// TIA Portal V18 export
// export: Created 2025-12-01T17:51:05.437198Z, ExportSetting None, DisplayName Totally Integrated Automation Portal, DisplayVersion V18 Update 5, DisplayName TIA Portal Openness, DisplayVersion V18 Update 5, DisplayName TIA Portal Teamcenter Gateway, DisplayVersion V18, DisplayName TIA Portal Version Control Interface, DisplayVersion V18, DisplayName STEP 7 Professional, DisplayVersion V18 Update 5, DisplayName STEP 7 Safety, DisplayVersion V18, DisplayName WinCC Professional, DisplayVersion V18 Update 5
FUNCTION "ST10Cyl_interface51-60" : Void   // FC1025, LAD
{ S7_Optimized_Access := 'FALSE' }
// stored: AutoNumber false, SetENOAutomatically false
   VAR_INPUT
      AlwaysON : Bool;
      E_stop : Bool;
   END_VAR
   VAR_TEMP
      tTest : Bool;
   END_VAR
   VAR_TEMP   // added for the SCL form of the ladder/FBD networks
      _w1 : Bool;
   END_VAR
BEGIN

REGION Network 1 (SCL): Cylinder 51-60 IO Interface (SCL)

   //Cylinder51 IO  L-UnloadingTransCylinder
   //Input
   "ST10Cylinder".Cy[51].In.WorkPositionSensor := "iL-UnloadingTransCylinderInWP";
   "ST10Cylinder".Cy[51].In.HomePositionSensor := "iL-UnloadingTransCylinderInHP";
   //Output
   "oL-UnloadingTransCylinderToWP" := "ST10Cylinder".Cy[51].Out.GoWorkPosition;
   "oL-UnloadingTransCylinderToHP" := "ST10Cylinder".Cy[51].Out.GoHomePosition;

   //Cylinder52 IO  L-UnloadingTransPalletLocationCylinder
   //Input
   "ST10Cylinder".Cy[52].In.WorkPositionSensor := "iL-UnloadingTransPalletLocationCylinderInWP";
   "ST10Cylinder".Cy[52].In.HomePositionSensor := "iL-UnloadingTransPalletLocationCylinderInHP";
   //Output
   "oL-UnloadingTransPalletLocationCylinderToWP" := "ST10Cylinder".Cy[52].Out.GoWorkPosition;
   "oL-UnloadingTransPalletLocationCylinderToHP" := "ST10Cylinder".Cy[52].Out.GoHomePosition;

   //Cylinder53 IO  L-UnloadingStopperCylinder1
   //Input
   "ST10Cylinder".Cy[53].In.WorkPositionSensor := "oL-UnloadingStopperCylinder1_ToWP";
   "ST10Cylinder".Cy[53].In.HomePositionSensor := "oL-UnloadingStopperCylinder1_ToHP";
   //Output
   "oL-UnloadingStopperCylinder1_ToWP" := "ST10Cylinder".Cy[53].Out.GoWorkPosition;
   "oL-UnloadingStopperCylinder1_ToHP" := "ST10Cylinder".Cy[53].Out.GoHomePosition;

   //Cylinder54 IO  L-UnloadingStopperCylinder2
   //Input
   "ST10Cylinder".Cy[54].In.WorkPositionSensor := "oL-UnloadingStopperCylinder2_ToWP";
   "ST10Cylinder".Cy[54].In.HomePositionSensor := "oL-UnloadingStopperCylinder2_ToHP";
   //Output
   "oL-UnloadingStopperCylinder2_ToWP" := "ST10Cylinder".Cy[54].Out.GoWorkPosition;
   "oL-UnloadingStopperCylinder2_ToHP" := "ST10Cylinder".Cy[54].Out.GoHomePosition;

   //Cylinder55 IO  L-UnloadingStopperCylinder3
   //Input
   "ST10Cylinder".Cy[55].In.WorkPositionSensor := "oL-UnloadingStopperCylinder3_ToWP";
   "ST10Cylinder".Cy[55].In.HomePositionSensor := "oL-UnloadingStopperCylinder3_ToHP";
   //Output
   "oL-UnloadingStopperCylinder3_ToWP" := "ST10Cylinder".Cy[55].Out.GoWorkPosition;
   "oL-UnloadingStopperCylinder3_ToHP" := "ST10Cylinder".Cy[55].Out.GoHomePosition;

   (*
   //Cylinder56  L-UnloadingStopperCylinder2_2
   //Input
   "ST10Cylinder".Cy[56].In.WorkPositionSensor := "oL-UnloadingStopperCylinder2_2";
   "ST10Cylinder".Cy[56].In.HomePositionSensor := NOT "oL-UnloadingStopperCylinder2_2";
   //Output
   "oL-UnloadingStopperCylinder2_2" := "ST10Cylinder".Cy[56].Out.GoWorkPosition;
   //"oI-0080TrayLoadingTraySupportCylinder1ToHP" := "ST10Cylinder".Cy[56].Out.GoHomePosition;

   //Cylinder57 L-UnloadingStopperCylinder3_1
   //Input
   "ST10Cylinder".Cy[57].In.WorkPositionSensor := "oL-UnloadingStopperCylinder3_1";
   "ST10Cylinder".Cy[57].In.HomePositionSensor := NOT "oL-UnloadingStopperCylinder3_1";
   //Output
   "oL-UnloadingStopperCylinder3_1" := "ST10Cylinder".Cy[57].Out.GoWorkPosition;
   //"oI-0070TrayLoadingTraySupportCylinder8ToHP" := "ST10Cylinder".Cy[57].Out.GoHomePosition;

   //Cylinder58 L-UnloadingStopperCylinder3_2
   //Input
   "ST10Cylinder".Cy[58].In.WorkPositionSensor := "oL-UnloadingStopperCylinder3_2";
   "ST10Cylinder".Cy[58].In.HomePositionSensor := NOT "oL-UnloadingStopperCylinder3_2";
   //Output
   "oL-UnloadingStopperCylinder3_2" := "ST10Cylinder".Cy[58].Out.GoWorkPosition;
   //"oI-0080TrayLoadingTrayLocationCylinderToHP" := "ST10Cylinder".Cy[58].Out.GoHomePosition;
   //

   *)
END_REGION

REGION Network 2: CY51 interface L-UnloadingTransCylinder
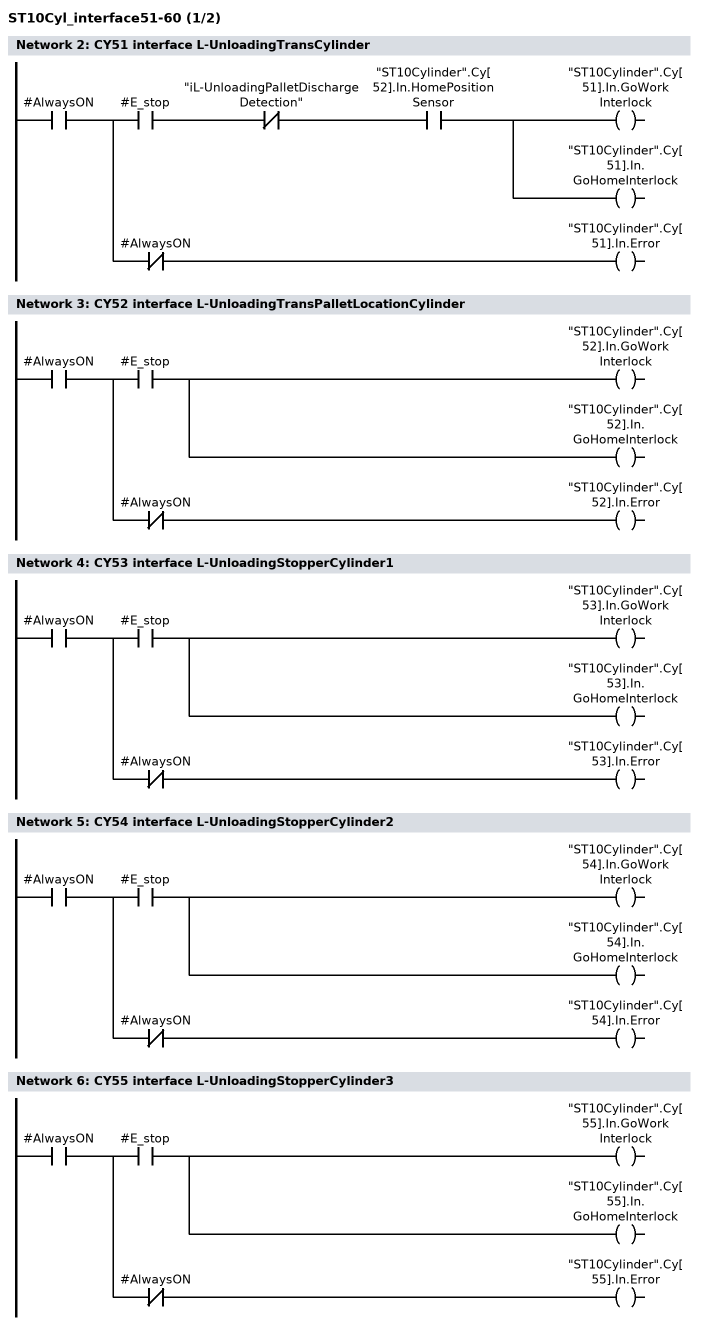
   RUNG wire#powerrail
      Contact( #AlwaysON )
      wire#w1
      Contact( #E_stop )
      I_Contact( "iL-UnloadingPalletDischargeDetection" )
      Contact( "ST10Cylinder".Cy[52].In.HomePositionSensor )
      wire#w2
      Coil( "ST10Cylinder".Cy[51].In.GoWorkInterlock )
   END_RUNG
   RUNG wire#w2
      Coil( "ST10Cylinder".Cy[51].In.GoHomeInterlock )
   END_RUNG
   RUNG wire#w1
      I_Contact( #AlwaysON )
      Coil( "ST10Cylinder".Cy[51].In.Error )
   END_RUNG
   // the same network as SCL:
   #_w1 := #AlwaysON AND #E_stop AND NOT "iL-UnloadingPalletDischargeDetection" AND "ST10Cylinder".Cy[52].In.HomePositionSensor;
   "ST10Cylinder".Cy[51].In.GoWorkInterlock := #AlwaysON AND #E_stop AND NOT "iL-UnloadingPalletDischargeDetection" AND "ST10Cylinder".Cy[52].In.HomePositionSensor;
   "ST10Cylinder".Cy[51].In.GoHomeInterlock := #_w1;
   "ST10Cylinder".Cy[51].In.Error := #AlwaysON AND NOT #AlwaysON;
END_REGION

REGION Network 3: CY52 interface L-UnloadingTransPalletLocationCylinder
   RUNG wire#powerrail
      Contact( #AlwaysON )
      wire#w1
      Contact( #E_stop )
      wire#w2
      Coil( "ST10Cylinder".Cy[52].In.GoWorkInterlock )
   END_RUNG
   RUNG wire#w2
      Coil( "ST10Cylinder".Cy[52].In.GoHomeInterlock )
   END_RUNG
   RUNG wire#w1
      I_Contact( #AlwaysON )
      Coil( "ST10Cylinder".Cy[52].In.Error )
   END_RUNG
   // the same network as SCL:
   "ST10Cylinder".Cy[52].In.GoWorkInterlock := #AlwaysON AND #E_stop;
   "ST10Cylinder".Cy[52].In.GoHomeInterlock := #AlwaysON AND #E_stop;
   "ST10Cylinder".Cy[52].In.Error := #AlwaysON AND NOT #AlwaysON;
END_REGION

REGION Network 4: CY53 interface L-UnloadingStopperCylinder1
   RUNG wire#powerrail
      Contact( #AlwaysON )
      wire#w1
      Contact( #E_stop )
      wire#w2
      Coil( "ST10Cylinder".Cy[53].In.GoWorkInterlock )
   END_RUNG
   RUNG wire#w2
      Coil( "ST10Cylinder".Cy[53].In.GoHomeInterlock )
   END_RUNG
   RUNG wire#w1
      I_Contact( #AlwaysON )
      Coil( "ST10Cylinder".Cy[53].In.Error )
   END_RUNG
   // the same network as SCL:
   "ST10Cylinder".Cy[53].In.GoWorkInterlock := #AlwaysON AND #E_stop;
   "ST10Cylinder".Cy[53].In.GoHomeInterlock := #AlwaysON AND #E_stop;
   "ST10Cylinder".Cy[53].In.Error := #AlwaysON AND NOT #AlwaysON;
END_REGION

REGION Network 5: CY54 interface L-UnloadingStopperCylinder2
   RUNG wire#powerrail
      Contact( #AlwaysON )
      wire#w1
      Contact( #E_stop )
      wire#w2
      Coil( "ST10Cylinder".Cy[54].In.GoWorkInterlock )
   END_RUNG
   RUNG wire#w2
      Coil( "ST10Cylinder".Cy[54].In.GoHomeInterlock )
   END_RUNG
   RUNG wire#w1
      I_Contact( #AlwaysON )
      Coil( "ST10Cylinder".Cy[54].In.Error )
   END_RUNG
   // the same network as SCL:
   "ST10Cylinder".Cy[54].In.GoWorkInterlock := #AlwaysON AND #E_stop;
   "ST10Cylinder".Cy[54].In.GoHomeInterlock := #AlwaysON AND #E_stop;
   "ST10Cylinder".Cy[54].In.Error := #AlwaysON AND NOT #AlwaysON;
END_REGION

REGION Network 6: CY55 interface L-UnloadingStopperCylinder3
   RUNG wire#powerrail
      Contact( #AlwaysON )
      wire#w1
      Contact( #E_stop )
      wire#w2
      Coil( "ST10Cylinder".Cy[55].In.GoWorkInterlock )
   END_RUNG
   RUNG wire#w2
      Coil( "ST10Cylinder".Cy[55].In.GoHomeInterlock )
   END_RUNG
   RUNG wire#w1
      I_Contact( #AlwaysON )
      Coil( "ST10Cylinder".Cy[55].In.Error )
   END_RUNG
   // the same network as SCL:
   "ST10Cylinder".Cy[55].In.GoWorkInterlock := #AlwaysON AND #E_stop;
   "ST10Cylinder".Cy[55].In.GoHomeInterlock := #AlwaysON AND #E_stop;
   "ST10Cylinder".Cy[55].In.Error := #AlwaysON AND NOT #AlwaysON;
END_REGION

REGION Network 7: CY56 interface
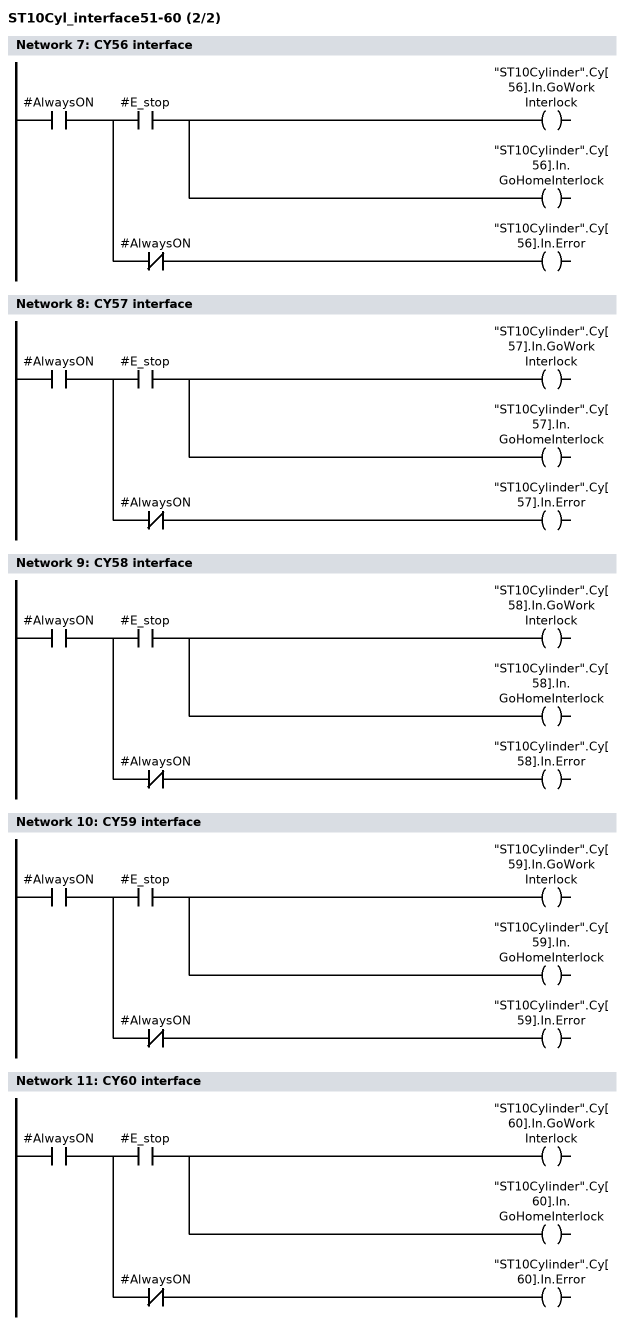
   RUNG wire#powerrail
      Contact( #AlwaysON )
      wire#w1
      Contact( #E_stop )
      wire#w2
      Coil( "ST10Cylinder".Cy[56].In.GoWorkInterlock )
   END_RUNG
   RUNG wire#w2
      Coil( "ST10Cylinder".Cy[56].In.GoHomeInterlock )
   END_RUNG
   RUNG wire#w1
      I_Contact( #AlwaysON )
      Coil( "ST10Cylinder".Cy[56].In.Error )
   END_RUNG
   // the same network as SCL:
   "ST10Cylinder".Cy[56].In.GoWorkInterlock := #AlwaysON AND #E_stop;
   "ST10Cylinder".Cy[56].In.GoHomeInterlock := #AlwaysON AND #E_stop;
   "ST10Cylinder".Cy[56].In.Error := #AlwaysON AND NOT #AlwaysON;
END_REGION

REGION Network 8: CY57 interface
   RUNG wire#powerrail
      Contact( #AlwaysON )
      wire#w1
      Contact( #E_stop )
      wire#w2
      Coil( "ST10Cylinder".Cy[57].In.GoWorkInterlock )
   END_RUNG
   RUNG wire#w2
      Coil( "ST10Cylinder".Cy[57].In.GoHomeInterlock )
   END_RUNG
   RUNG wire#w1
      I_Contact( #AlwaysON )
      Coil( "ST10Cylinder".Cy[57].In.Error )
   END_RUNG
   // the same network as SCL:
   "ST10Cylinder".Cy[57].In.GoWorkInterlock := #AlwaysON AND #E_stop;
   "ST10Cylinder".Cy[57].In.GoHomeInterlock := #AlwaysON AND #E_stop;
   "ST10Cylinder".Cy[57].In.Error := #AlwaysON AND NOT #AlwaysON;
END_REGION

REGION Network 9: CY58 interface
   RUNG wire#powerrail
      Contact( #AlwaysON )
      wire#w1
      Contact( #E_stop )
      wire#w2
      Coil( "ST10Cylinder".Cy[58].In.GoWorkInterlock )
   END_RUNG
   RUNG wire#w2
      Coil( "ST10Cylinder".Cy[58].In.GoHomeInterlock )
   END_RUNG
   RUNG wire#w1
      I_Contact( #AlwaysON )
      Coil( "ST10Cylinder".Cy[58].In.Error )
   END_RUNG
   // the same network as SCL:
   "ST10Cylinder".Cy[58].In.GoWorkInterlock := #AlwaysON AND #E_stop;
   "ST10Cylinder".Cy[58].In.GoHomeInterlock := #AlwaysON AND #E_stop;
   "ST10Cylinder".Cy[58].In.Error := #AlwaysON AND NOT #AlwaysON;
END_REGION

REGION Network 10: CY59 interface
   RUNG wire#powerrail
      Contact( #AlwaysON )
      wire#w1
      Contact( #E_stop )
      wire#w2
      Coil( "ST10Cylinder".Cy[59].In.GoWorkInterlock )
   END_RUNG
   RUNG wire#w2
      Coil( "ST10Cylinder".Cy[59].In.GoHomeInterlock )
   END_RUNG
   RUNG wire#w1
      I_Contact( #AlwaysON )
      Coil( "ST10Cylinder".Cy[59].In.Error )
   END_RUNG
   // the same network as SCL:
   "ST10Cylinder".Cy[59].In.GoWorkInterlock := #AlwaysON AND #E_stop;
   "ST10Cylinder".Cy[59].In.GoHomeInterlock := #AlwaysON AND #E_stop;
   "ST10Cylinder".Cy[59].In.Error := #AlwaysON AND NOT #AlwaysON;
END_REGION

REGION Network 11: CY60 interface
   RUNG wire#powerrail
      Contact( #AlwaysON )
      wire#w1
      Contact( #E_stop )
      wire#w2
      Coil( "ST10Cylinder".Cy[60].In.GoWorkInterlock )
   END_RUNG
   RUNG wire#w2
      Coil( "ST10Cylinder".Cy[60].In.GoHomeInterlock )
   END_RUNG
   RUNG wire#w1
      I_Contact( #AlwaysON )
      Coil( "ST10Cylinder".Cy[60].In.Error )
   END_RUNG
   // the same network as SCL:
   "ST10Cylinder".Cy[60].In.GoWorkInterlock := #AlwaysON AND #E_stop;
   "ST10Cylinder".Cy[60].In.GoHomeInterlock := #AlwaysON AND #E_stop;
   "ST10Cylinder".Cy[60].In.Error := #AlwaysON AND NOT #AlwaysON;
END_REGION
END_FUNCTION
